// TIA Portal V17 export
// export: Created 2024-08-07T21:43:59.6367971Z, ExportSetting WithDefaults, DisplayName Totally Integrated Automation Portal, DisplayVersion V17 Update 7, DisplayName TIA Portal Openness, DisplayVersion V17 Update 7, DisplayName TIA Portal Version Control Interface, DisplayVersion V17, DisplayName SINAMICS Startdrive Advanced, DisplayVersion V17 SP2, DisplayName SINAMICS Startdrive G110M, G120, G120C, G120D, G120P, G115D, DisplayVersion V17 SP2, DisplayName SINAMICS Startdrive G130, G150, S120, S150, SINAMICS MV, S210, DisplayVersion V17 SP2, DisplayName STEP 7 Professional, DisplayVersion V17 Update 7, DisplayName STEP 7 Safety, DisplayVersion V17 Update 6, DisplayName WinCC Advanced / Unified PC, DisplayVersion V17 Update 7
DATA_BLOCK "DB_INST_READINGS"   // DB300
VERSION : 0.1
// stored: AutoNumber false, DBAccessibleFromOPCUA true, DBAccessibleFromWebserver true, InstanceOfName FB_READINGS, InstanceOfType FB
"FB_READINGS"
   // VAR
   //    Reading : Array[1.."MaxDataReading"] of Struct
   //       Done : Bool;
   //       OK : Bool;
   //       NOK : Bool;
   //       Scan : String[70];
   //       NFP : String[30];
   //       IJC : Array[1.."NumberOfmessages"] of Struct
   //          SendMsg : Bool;
   //          Done : Bool;
   //          Answer : Int;
   //          State : USInt;
   //       END_STRUCT;
   //    END_STRUCT;
   //    ReadingsDone : Bool;
   //    Errors : Array[1..2] of Word;
   // END_VAR
BEGIN
END_DATA_BLOCK
